# EPICS substitutions: Db/fru_atca_rtm_lcls.substitutions
#==============================================================================
# Abs:  ATCA RTM FRU PV subset
#
# Name:  fru_atca_rtm_lcls.substitutions
#
# Macros in:
#	dev      Shelf name, for example CRAT:LI28:RF01
#	prefix   String in PV name that identifies the FRU sensor is associated with (if there is one)
#		 PV name syntax: $(dev):$(prefix)$(attr)$(sensinst)
#		 For atca systems, prefix is "<frutype><instance>_", for example FB1_ for the first FB
#		 or CU2_ for the second cooling unit
#		 For supermicro, the sensors are not associated with a FRU, so prefix is an empty string
#	aliasprefix Temporary string to keep PV names backward-compatible via alias
#	id       String identifier, for example 'CU' for cooling unit
#       unit     Instance of this type of module, for example 2 for the second MCH in a carrier
#       attr	 Used in PV attribute, for example FAN1SPEED or TEMP2
#       sensinst Instance of this type of sensor on this module
#       type     Sensor type code, defined in IPMI spec (and src/ipmiDef.h)
#       fruid    FRU ID according to MicroTCA spec
#	dev      Shelf name, for example CRAT:LI28:RF01
#	cod      String identifier, for example 'CU' for cooling unit
#       inst     Instance of this type of module, for example 2 for the second MCH in a carrier
#       attr	 Used in PV attribute, for example FAN1SPEED or TEMP2
#       sensinst Instance of this type of sensor on this module
#       type     Sensor type code, defined in IPMI spec (and src/ipmiDef.h)
#       fruid    FRU ID according to MicroTCA spec
#
#==============================================================================
#

file fru_common.db
{
   pattern { dev	, id		, unit		, fruid		}
           { $(dev)	, $(id)		, $(unit)  	, $(fruid)	}
}

file sensor_ai.db
{
   pattern { dev	, prefix	, aliasprefix	,  attr		, sensinst	, type	, fruid }
           { $(dev)	, $(id)$(unit):	, $(id)$(unit)_	,  TEMP		, 1		, 1	, $(fruid)	}
           { $(dev)	, $(id)$(unit):	, $(id)$(unit)_	,  TEMP		, 2		, 1	, $(fruid)	}
           { $(dev)	, $(id)$(unit):	, $(id)$(unit)_	,  V		, 1		, 2	, $(fruid)	}
           { $(dev)	, $(id)$(unit):	, $(id)$(unit)_	,  V		, 2		, 2	, $(fruid)	}
           { $(dev)	, $(id)$(unit):	, $(id)$(unit)_	,  I		, 1		, 3	, $(fruid)	}
           { $(dev)	, $(id)$(unit):	, $(id)$(unit)_	,  I		, 2		, 3	, $(fruid)	}
}
